{attribute 'GeneratedUsingTerminal: EP2816-0003-0016'}
{attribute addProperty BoxType "EP2816-0003-0016"}
{attribute addProperty Id "Diag_InputAT %I*ARRAY[0..7] OF BOOL8"}
{attribute addProperty CRC "568896300"}
{attribute addProperty Size "8"}
TYPE DIG_Diag_Inputs_Channel_584303BF EXTENDS InputBase_8311D824 :
STRUCT
	{attribute addProperty Name "Diag_Input"}
	Diag_Input AT %I* : ARRAY[0..7] OF BOOL;
END_STRUCT
END_TYPE

(* stored: Version 1.2.0.0, ProductVersion 3.1.4024.11
   DUT DIG_Diag_Inputs_Channel_584303BF: Id {ce43d2e9-2a4f-4258-a902-27895fec0514} *)
